# B&R Automation Studio project AS_lab_3
Automation Studio 4.5.2.102

## Configuration Real

CPU 4PP065.0571-P74, AutomationRuntime D4.52, Build 4.1.2, Vc V4.52.0, Safety 1.6

### Task classes (Cpu.sw)
```
Cyclic#1 (cycle 2000 us):
  SDCAxisCtr <- SDCAxisCtrlX.prg
DataObjects: Acp10sys
NcDataObjects: acp10etxen <- acp10etxen.dob, Axis_Xa <- Axis_Xobj.Axis_Xa.dob, Axis_Xi <- Axis_Xobj.Axis_Xi.dob
VcDataObjects: GUI <- GUI.dob
Binaries: TCData, udbdef, ashwd, Role, User, sysconf, ashwac, asfw, arconfig, iomap, Acp10map, acp10cfg
Libraries: Acp10man, Acp10par, NcGlobal, Acp10sdc, AsBrStr, Acp10_MC, brsystem, sys_lib, runtime, Acp10sim, AsIOTime, MotorCtrl, astime, fileio, powerlnk
```

### Hardware
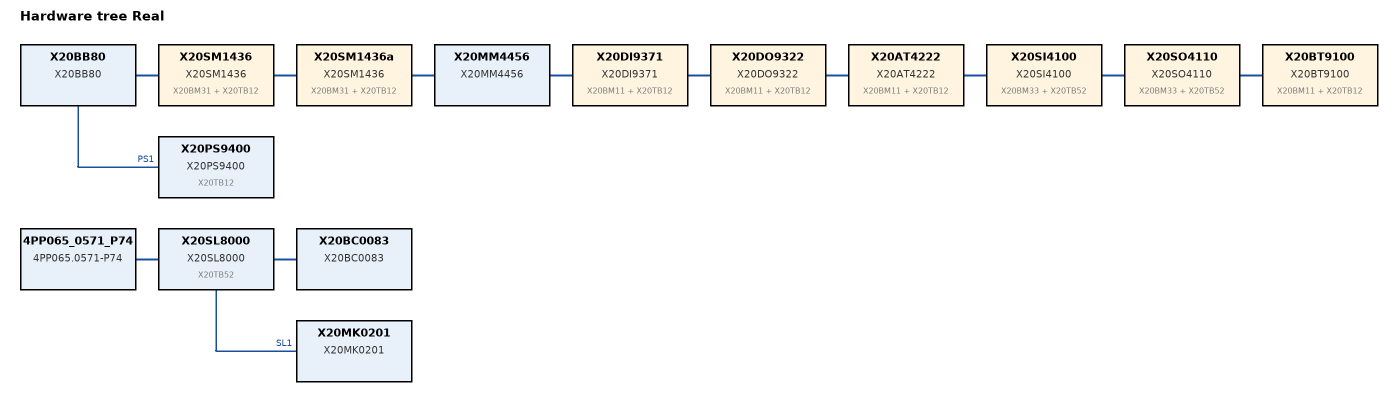
```
4PP065_0571_P74 : 4PP065.0571-P74 v1.1.2.0
  Connector IF5:
    ActivateDevice = 1
    Mode = Manual
    InternetAddress = 10.0.1.10
    SubnetMask = 255.255.255.0
  ConfigurationID = labBR
  TimerDeviceType = EPLX2X
  TimerDevice = 4PP065_0571_P74.IF4
  TaskClassIdleTime = 2000
  Cyclic1Duration = 2000
  Cyclic1Output = 1
  VcObjectName = GUI
X20AT4222 : X20AT4222 v1.2.3.0  [SS1 -> X20TB12e.SS; SL -> X20BM11b.SL1]
X20BB80 : X20BB80 v1.0.2.0
X20BC0083 : X20BC0083 v2.8.0.0  [PLK1 -> X20SL8000.PLK2 [Cable Type=PowerlinkCable, Length=10, Version=1.0.0.2]; SL -> X20BB80.SL1]
X20BM11 : X20BM11 v1.0.0.1  [X2X1 -> X20MM4456.X2X2]
X20BM11a : X20BM11 v1.0.0.1  [X2X1 -> X20BM11.X2X2]
X20BM11b : X20BM11 v1.0.0.1  [X2X1 -> X20BM11a.X2X2]
X20BM11c : X20BM11 v1.0.0.1  [X2X1 -> X20BM33a.X2X2]
X20BM31 : X20BM31 v1.0.0.1  [X2X1 -> X20BB80.IF1]
X20BM31a : X20BM31 v1.0.0.1  [X2X1 -> X20BM31.X2X2]
X20BM33 : X20BM33 v1.0.0.4  [X2X1 -> X20BM11b.X2X2]
X20BM33a : X20BM33 v1.0.0.4  [X2X1 -> X20BM33.X2X2]
X20BT9100 : X20BT9100 v1.0.3.0  [SS1 -> X20TB12f.SS; SL -> X20BM11c.SL1]
X20DI9371 : X20DI9371 v1.0.2.0  [SS1 -> X20TB12c.SS; SL -> X20BM11.SL1]
X20DO9322 : X20DO9322 v1.0.3.0  [SS1 -> X20TB12d.SS; SL -> X20BM11a.SL1]
X20MK0201 : X20MK0201 v1.0.0.0  [SL -> X20SL8000.SL1]
X20MM4456 : X20MM4456 v1.1.5.0  [X2X1 -> X20BM31a.X2X2]
X20PS9400 : X20PS9400 v1.0.2.4  [SS1 -> X20TB12.SS; PS -> X20BB80.PS1]
X20SI4100 : X20SI4100 v1.10.1.1  [SS1 -> X20TB52a.SS; SL -> X20BM33.SL1]
X20SL8000 : X20SL8000 v1.6.5.1  [PLK1 -> 4PP065_0571_P74.IF4 [Cable Type=PowerlinkCable, Length=10, Version=1.0.0.2]; PLK2 -> X20BC0083.PLK1 [Cable Type=PowerlinkCable, Length=10, Version=1.0.0.2]; SS1 -> X20TB52.SS]
  SafeProject = SafeLOGIC-1
X20SM1436 : X20SM1436 v1.4.2.1  [SS1 -> X20TB12a.SS; SL -> X20BM31.SL1]
X20SM1436a : X20SM1436 v1.4.2.1  [SS1 -> X20TB12b.SS; SL -> X20BM31a.SL1]
X20SO4110 : X20SO4110 v1.10.1.1  [SS1 -> X20TB52b.SS; SL -> X20BM33a.SL1]
  SafeModuleID = 3
X20TB12 : X20TB12 v1.0.0.0
X20TB12a : X20TB12 v1.0.0.0
X20TB12b : X20TB12 v1.0.0.0
X20TB12c : X20TB12 v1.0.0.0
X20TB12d : X20TB12 v1.0.0.0
X20TB12e : X20TB12 v1.0.0.0
X20TB12f : X20TB12 v1.0.0.0
X20TB52 : X20TB52 v1.0.0.1
X20TB52a : X20TB52 v1.0.0.1
X20TB52b : X20TB52 v1.0.0.1
```

### IoMap.iom - 4PP065_0571_P74/IoMap.iom
```iecst
VAR_CONFIG
	::SDCAxisCtr:pwm_period AT %QW."X20MM4456".PeriodDurationPWM;
	::SDCAxisCtr:axis_X.pwm_value AT %QW."X20MM4456".PulseWidthCurrentPWM01;
	::SDCAxisCtr:axis_X.reset_error AT %QX."X20MM4456".ClearError01;
	::SDCAxisCtr:axis_X.reset_counter AT %QX."X20MM4456".ResetCounter01;
	::SDCAxisCtr:axis_X.counter AT %IW."X20MM4456".Counter01;
	::SDCAxisCtr:axis_X.endswitch_a_reached AT %IX."X20MM4456".StatusInput03;
	::SDCAxisCtr:axis_X.endswitch_b_reached AT %IX."X20MM4456".StatusInput04;
	::SDCAxisCtr:coil_pwm_value AT %QW."X20MM4456".PulseWidthCurrentPWM04;
END_VAR
```

### Acp10map1.ncm - 4PP065_0571_P74/Motion/Acp10map1.ncm
```
NcMapping (NcSwId=ACP10, DisabledNodesAreHidden=False)
  NcObject Axis_X (ModuleAddress=SDC_IF1.ST2, InterfaceType=SDC, Type=ncAXIS, Channel=1, InitParameter=Axis_Xi, AcoposParameter=Axis_Xa, Disabled=FALSE, ModuleDisabled=FALSE)
```

### Acp10map.ncm - 4PP065_0571_P74/Package/Acp10map.ncm
```
NcMapping (NcSwId=Acp10)
  NcObject X20SM1436_ncAXIS1 (ModuleId=X20SM1436, ModuleAddress=SDC_IF1.ST1, Type=ncAXIS, Channel=1, AcoposSimulation=Off, Disabled=TRUE, ModuleDisabled=FALSE)
  NcObject X20SM1436a_ncAXIS1 (ModuleId=X20SM1436a, ModuleAddress=SDC_IF1.ST2, Type=ncAXIS, Channel=1, AcoposSimulation=Off, Disabled=TRUE, ModuleDisabled=FALSE)
  NcObject 8I64xxxxxxx.00x-1_ncAXIS1 (ModuleId=8I64xxxxxxx.00x-1, ModuleAddress=SDC_IF1.ST3, Type=ncAXIS, Channel=1, AcoposSimulation=Off, Disabled=TRUE, ModuleDisabled=FALSE)
```

## Logical view

Binary libraries used (declarations not repeated): operator, runtime, astime, AsIecCon, Acp10man, Acp10par, NcGlobal, Acp10sdc, AsBrStr, Acp10_MC, brsystem, sys_lib, Acp10sim, AsIOTime

### Global.var - Global variables
```iecst
VAR
	Axis_X : ACP10AXIS_typ;
	Axis_X_HW : SdcHwCfg_typ;
	Axis_X_EncIf : SdcEncIf16_typ;
	Axis_X_DrvIf : SdcDrvIf16_typ;
	Axis_X_DiDoIf : SdcDiDoIf_typ;
END_VAR
```

### Package Logical/Libraries - Global libraries

### Library Logical/Libraries/MotorCtrl (ANSIC)

#### MotorCtrl.fun
```iecst
FUNCTION_BLOCK FB_Regulator
	VAR_INPUT
		e : REAL;
		e_prev : REAL;
	END_VAR
	VAR_OUTPUT
		u : REAL;
	END_VAR
	VAR
		u_raw : REAL;
		k_p : REAL;
		k_i : REAL;
		integrator : FB_Integrator;
		iyOld : REAL;
		max_abs_value : REAL;
	END_VAR
END_FUNCTION_BLOCK

FUNCTION_BLOCK FB_Motor
	VAR_INPUT
		u : REAL;
	END_VAR
	VAR_OUTPUT
		w : REAL;
		phi : REAL;
	END_VAR
	VAR
		integrator : FB_Integrator;
		integrator_phi : FB_Integrator;
		Tm : REAL;
		ke : REAL;
		enable_reg : BOOL;
	END_VAR
END_FUNCTION_BLOCK

FUNCTION_BLOCK FB_Integrator
	VAR_INPUT
		in : REAL;
	END_VAR
	VAR_OUTPUT
		out : REAL;
	END_VAR
	VAR
		dt : REAL;
		direct : BOOL;
	END_VAR
END_FUNCTION_BLOCK

FUNCTION_BLOCK FB_Axis
	VAR_INPUT
		u : REAL;
		force_a : BOOL;
		force_b : BOOL;
		endswitch_a_reached : BOOL;
		endswitch_b_reached : BOOL;
	END_VAR
	VAR_OUTPUT
		reset_error : BOOL;
		reset_counter : BOOL;
		pwm_value : INT;
		counter : INT;
		speed : INT;
	END_VAR
	VAR
		last_counter : INT;
		ForceStop : BOOL;
		Home : BOOL;
	END_VAR
END_FUNCTION_BLOCK
```

#### FB_Axis.c
```c
#include <bur/plctypes.h>
#ifdef __cplusplus
	extern "C"
	{
#endif
#include "MotorCtrl.h"
#ifdef __cplusplus
	};
#endif
/* TODO: Add your comment here */
void FB_Axis(struct FB_Axis* inst)
{
	if (inst->Home)
	{
		inst->pwm_value = 0;
		inst->reset_counter = 1;
		inst->Home = 0;
	}

	if (!inst->ForceStop)
	{
		if (inst->endswitch_a_reached && inst->u < 0)
		{
			inst->pwm_value = 0;
			inst->reset_error = 1;
		}
		else if (inst->endswitch_b_reached && inst->u > 0)
		{
			inst->pwm_value = 0;
			inst->reset_error = 1;
		}
		else if (inst->force_a)
		{
			inst->pwm_value = 0;
			inst->endswitch_a_reached = inst->force_a;
		}
		else if (inst->force_b)
		{
			inst->pwm_value = 0;
			inst->endswitch_b_reached = inst->force_b;
		}
		else
		{
			inst->pwm_value = inst->u / 24.0 * 32767;
			inst->reset_error = 0;
		}
	}
	else
	{
		inst->pwm_value = 0;
	}

	inst->speed = inst->u / 24.0 * 6500;
}
```

#### FB_Regulator.c
```c
#include <bur/plctypes.h>
#ifdef __cplusplus
	extern "C"
	{
#endif
#include "MotorCtrl.h"
#ifdef __cplusplus
	};
#endif

#include "Math.h"
/* TODO: Add your comment here */
void FB_Regulator(struct FB_Regulator* inst)
{
	if (inst->integrator.direct)
		inst->integrator.in = inst->k_i * inst->e_prev + inst->iyOld / inst->integrator.dt;
	else
		inst->integrator.in = inst->k_i * inst->e + inst->iyOld / inst->integrator.dt;
	FB_Integrator(&inst->integrator);
	inst->u_raw = (fabs(inst->k_p * inst->e) < inst->max_abs_value ? inst->k_p * inst->e : inst->max_abs_value * copysign(1.0, inst->k_p * inst->e)) +
		inst->integrator.out;
	inst->u = fabs(inst->u_raw) < inst->max_abs_value ? inst->u_raw : inst->max_abs_value * copysign(1.0, inst->u_raw);
	inst->iyOld = inst->u - inst->u_raw;
}
```

### Package Logical/Axis_Xobj - Axis_Xobj

### Axis_Xi.ax
```
InitParameter (Version=5.02.1, NcSwId=Acp10)
  ACP10AXIS_typ:
    dig_in:
      level:
        reference = ncACTIV_HI
        pos_hw_end = ncACTIV_HI
        neg_hw_end = ncACTIV_HI
        trigger1 = ncACTIV_HI
        trigger2 = ncACTIV_LO + ncQUICKSTOP
    encoder_if:
      parameter:
        count_dir = ncSTANDARD
        scaling:
          load:
            units = 3000
            rev_motor = 1
    limit:
      parameter:
        v_pos = 10000
        v_neg = 10000
        a1_pos = 10000.0
        a2_pos = 10000.0
        a1_neg = 10000.0
        a2_neg = 10000.0
        t_jolt = 0
        t_in_pos = 0
        pos_sw_end = 2000000000
        neg_sw_end = -2000000000
        ds_warning = 500
        ds_stop = 50000.0
        a_stop = 1.0e30
        dv_stop = 0
        dv_stop_mode = ncOFF
    controller:
      mode = ncPOSITION
      position:
        kv = 10.0
        tn = 0
        t_predict = 0.0004
        t_total = 0.0004
        p_max = 1.0e30
        i_max = 0
      speed:
        kv = 2.0
        tn = 0
        t_filter = 0.0
        isq_filter1:
          type = ncOFF
          a0 = 0.0
          a1 = 0.0
          b0 = 0.0
          b1 = 0.0
          b2 = 0.0
          c0_par_id = 0
          c1_par_id = 0
        isq_filter2:
          type = ncOFF
          a0 = 0.0
          a1 = 0.0
          b0 = 0.0
          b1 = 0.0
          b2 = 0.0
          c0_par_id = 0
          c1_par_id = 0
        isq_filter3:
          type = ncOFF
          a0 = 0.0
          a1 = 0.0
          b0 = 0.0
          b1 = 0.0
          b2 = 0.0
          c0_par_id = 0
          c1_par_id = 0
      uf:
        type = ncLINEAR + ncCORRECTION
        auto_config = ncMOTOR_PAR
        u0 = 0
        un = 0
        fn = 50.0
        k_f_slip = 0
      ff:
        torque_load = 0.0
        torque_pos = 0.0
        torque_neg = 0.0
        kv_torque = 0.0
        inertia = 0.0
        t_filter_a = 0.0
    move:
      stop:
        parameter[0]:
          decel_ramp = ncA_LIMIT
          controller = ncON
        parameter[1]:
          decel_ramp = ncA_LIMIT
          controller = ncON
        parameter[2]:
          decel_ramp = ncA_LIMIT
          controller = ncON
        parameter[3]:
          decel_ramp = ncA_LIMIT
          controller = ncON
        quickstop:
          decel_ramp = ncA_LIMIT
          t_jolt = 0
        drive_error:
          decel_ramp = ncA_LIMIT
      homing:
        parameter:
          s = 0
          v_switch = 6000.0
          v_trigger = 2000.0
          a = 10000.0
          mode = ncEND_SWITCH
          edge_sw = ncNEGATIVE
          start_dir = ncPOSITIVE
          trigg_dir = ncNEGATIVE
          ref_pulse = ncOFF
          fix_dir = ncOFF
          tr_s_block = 0
          torque_lim = 0
          ds_block = 0
          ds_stop = 0
      basis:
        parameter:
          v_pos = 5000
          v_neg = 5000
          a1_pos = 50000
          a2_pos = 50000
          a1_neg = 50000
          a2_neg = 50000
    message:
      text:
        parameter:
          format = ncBREAK
          columns = 80
          data_modul = acp10etxen
```

### Program Logical/SDCAxisCtrlX (ANSIC)

#### Variables.var
```iecst
VAR
	axis_X : FB_Axis;
	CoilPowered : BOOL;
	CoilPWM : INT;
	fb_regulator : FB_Regulator;
	PWM_Period : UINT;
END_VAR
```

#### Main.c
```c
/*#include <bur/plctypes.h>
#include <math.h>

#ifdef _DEFAULT_INCLUDES
	#include <AsDefault.h>
#endif

#define MOTORS_COUNT 3

void _INIT MainINIT(void)
{
	//Устанавливаем типы SDC модулей
	Axis_X_HW.EncIf1_Typ = ncSDC_ENC16;
	Axis_X_HW.DiDoIf_Typ = ncSDC_DIDO;
	Axis_X_HW.DrvIf_Typ = ncSDC_DRVSERVO16;
	//Устанавливаем имена переменных
	strcpy(Axis_X_HW.EncIf1_Name, "Axis_X_EncIf");
	strcpy(Axis_X_HW.DrvIf_Name, "Axis_X_DrvIf");
	strcpy(Axis_X_HW.DiDoIf_Name, "Axis_X_DiDoIf");
	//Устанавливаем входы готовности и нормальной
	работы
	Axis_X_EncIf.iEncOK = 1;
	Axis_X_DrvIf.iDrvOK = 1;
	Axis_X_DrvIf.iStatusEnable = 1;
	Axis_X_DiDoIf.iDriveReady = 1;

	Axis_X_EncIf.iLifeCnt++;
	Axis_X_DiDoIf.iLifeCntDriveEnable++;
	Axis_X_DiDoIf.iLifeCntDriveReady++;
	Axis_X_DiDoIf.iLifeCntNegHwEnd++;
	Axis_X_DiDoIf.iLifeCntPosHwEnd++;
	Axis_X_DiDoIf.iLifeCntReference++;
	Axis_X_DrvIf.iLifeCnt++;
	Axis_X_EncIf.iActTime = (INT)AsIOTimeCyclicStart();

	int i = 0;
	for (; i < MOTORS_COUNT; i++)
	{
		motors[i].pwm_value = 0;
		motors[i].pwm_percentage = 0;
		motors[i].counter = 0;
		motors[i].coordinate = 0;
		motors[i].button_status = 0;
		motors[i].reset_error = 0;
		motors[i].endswitch_a_reached = 0;
		motors[i].endswitch_b_reached = 0;
	}
	pwm_period = 200;
	coil_powered = 0;
	coil_pwm_value = 0;
	emergency_stop = 0;
	current_motor_index = 0;

	check = 0;
	a = 0;
	n = 0;
}

void _CYCLIC MainCYCLIC(void)
{
	int i = 0, j = 0;
	if (emergency_stop)  //аварийная остановка
	{
		for (i = 0; i < MOTORS_COUNT; i++)
		{
			motors[i].pwm_value = 0;
			motors[i].pwm_percentage = 0;
		}
		coil_powered = 0;
		check = 0;
		emergency_stop = 0;
	}
	current_motor = &motors[current_motor_index];
	for (i = 0; i < MOTORS_COUNT; i++)  //цикл для обозначения на экране текущей степени (кнопка подсвечивается белым цветом)
	{
		MotorFunctionBlock(&motors[i]);
		if (current_motor == &motors[i])
		{
			motors[i].button_status = 1 << 1;
		}
		else
		{
			motors[i].button_status = 0;
		}
	}
	if (coil_powered)  //проверяем напряжение на катушке
	{
		coil_pwm_value = 32767;
		if (check)
		{
			switch (mode)  //проверяем выбранный режим
			{
				case 1:
					switch (path)  //проверяем выбранный контур, разбиваем его и заполняем массив координат соответствующими значениями
					{
						case 1:
							for (i = 0; i < 20; i++)
							{
								coordX[i] = 150 * pi * i / (10*sqrt(2));
								coordY[i] = 150 * pi * i / (10*sqrt(2));
								coordZ[i] = 250 * sin(sqrt(coordX[i] * coordX[i] + coordY[i] * coordY[i]) / 150);
							}
							break;
						case 2:
							for (i = 0; i < 20; i++)
							{
								coordX[i] = 30 * i;
								coordY[i] = 30 * i;
								coordZ[i] = (coordX[i] * coordX[i] + coordY[i] * coordY[i]) / 180;
							}
							break;
						case 0:
							break;
					}
					distX = coordX[a+1] - coordX[a];  //длина полученных отрезков
					distY = coordY[a+1] - coordY[a];
					distZ = coordZ[a+1] - coordZ[a];
					if ((fabs(distX) >= fabs(distY)) && (fabs(distX) >= fabs(distZ)))  //поиск наибольшей проекции каждого отрезка
					{
						index[a] = 2;
					}
					if ((fabs(distY) >= fabs(distX)) && (fabs(distY) >= fabs(distZ)))
					{
						index[a] = 0;
					}
					if ((fabs(distZ) >= fabs(distX)) && (fabs(distZ) >= fabs(distY)))
					{
						index[a] = 1;
					}
					if (index[a] == 2)  //проекция на ось X наибольшая
					{
						if (motors[2].counter > coordX[a+1])  //если степень находится за следующей точкой, то двигаем её в обратном направлении
						{
							motors[2].pwm_percentage_float = -50.0;
						}
						if (motors[2].counter < coordX[a+1])  //если перед точкой, то в прямом направлении
						{
							motors[2].pwm_percentage_float = 50.0;
						}
						motors[0].pwm_percentage_float = (distY * motors[2].pwm_percentage_float) / distX;  //вычисляем реальное значение ШИМ (в процентах)
						motors[1].pwm_percentage_float = (distZ * motors[2].pwm_percentage_float) / distX;
						if ((motors[2].counter >= (coordX[a+1] - 2)) && (motors[2].counter <= (coordX[a+1] + 2)))
						{
							if (a < 18)  //проверка пройденных точек
							{
								a++;
							}
							else  //если все точки пройдены, то отключаем степени и сбрасываем выбранные режим и контур
							{
								for (i = 0; i < MOTORS_COUNT; i++)
								{
									motors[i].pwm_percentage_float = 0.0;
									motors[i].pwm_value_float = 0.0;
									motors[i].pwm_percentage = 0;
									motors[i].pwm_value = 0;
								}
								check = 0;
								mode = 0;
								path = 0;
								a = 0;
							}
						}
					}
					if (index[a] == 0)  //проекция на ось Y максимальная
					{
						if (motors[0].counter > coordY[a+1])  //если степень находится за следующей точкой, то двигаем её в обратном направлении
						{
							motors[0].pwm_percentage_float = -50.0;
						}
						if (motors[0].counter < coordY[a+1])  //если перед точкой, то в прямом направлении
						{
							motors[0].pwm_percentage_float = 50.0;
						}
						motors[2].pwm_percentage_float = (distX * motors[0].pwm_percentage_float) / distY;  //вычисляем реальное значение ШИМ (в процентах)
						motors[1].pwm_percentage_float = (distZ * motors[0].pwm_percentage_float) / distY;
						if ((motors[0].counter >= (coordY[a+1] - 2)) && (motors[0].counter <= (coordY[a+1] + 2)))
						{
							if (a < 18)  //проверка пройденных точек
							{
								a++;
							}
							else  //если все точки пройдены, то отключаем степени и сбрасываем выбранные режим и контур
							{
								for (i = 0; i < MOTORS_COUNT; i++)
								{
									motors[i].pwm_percentage_float = 0.0;
									motors[i].pwm_value_float = 0.0;
									motors[i].pwm_percentage = 0;
									motors[i].pwm_value = 0;
								}
								check = 0;
								mode = 0;
								path = 0;
								a = 0;
							}
						}
					}
					if (index[a] == 1)  //проекция на ось Z максимальная
					{
						if (motors[1].counter > coordZ[a+1])  //если степень находится за следующей точкой, то двигаем её в обратном направлении
						{
							motors[1].pwm_percentage_float = -50.0;
						}
						if (motors[1].counter < coordZ[a+1])  //если перед точкой, то в прямом направлении
						{
							motors[1].pwm_percentage_float = 50.0;
						}
						motors[2].pwm_percentage_float = (distX * motors[1].pwm_percentage_float) / distZ;  //вычисляем реальное значение ШИМ (в процентах)
						motors[0].pwm_percentage_float = (distY * motors[1].pwm_percentage_float) / distZ;
						if ((motors[1].counter >= (coordZ[a+1] - 2)) && (motors[1].counter <= (coordZ[a+1] + 2)))
						{
							if (a < 18)  //проверка пройденных точек
							{
								a++;
							}
							else  //если все точки пройдены, то отключаем степени и сбрасываем выбранные режим и контур
							{
								for (i = 0; i < MOTORS_COUNT; i++)
								{
									motors[i].pwm_percentage_float = 0.0;
									motors[i].pwm_value_float = 0.0;
									motors[i].pwm_percentage = 0;
									motors[i].pwm_value = 0;
								}
								check = 0;
								mode = 0;
								path = 0;
								a = 0;
							}
						}
					}
					for (i = 0; i < MOTORS_COUNT; i++)
					{
						motors[i].pwm_percentage = motors[i].pwm_percentage_float;  //присваиваем значению ШИМ на слайдере на экране к реальному значению ШИМ (для наглядности)
					}
					for (i = 0; i < MOTORS_COUNT; i++)
					{
						motors[i].pwm_value_float = 32767 * motors[i].pwm_percentage_float / 100;  //вычисляем ШИМ для каждой степени
						motors[i].pwm_value = motors[i].pwm_value_float;  //приводим значение типа REAL к значению типа INT и пересылаем на двигатель
						if ((!motors[i].endswitch_a_reached) && (!motors[i].endswitch_b_reached))
						{
							motors[i].reset_error = 0;
						}
						if ((motors[i].endswitch_a_reached) && (motors[i].pwm_percentage > 0))  //если достигнут концевой датчик, то останавливаем все степени и сбрасываем ошибку
						{
							motors[i].reset_error = 1;
							for (j = 0; j < MOTORS_COUNT; j++)
							{
								motors[j].pwm_percentage_float = 0.0;
								motors[j].pwm_value_float = 0.0;
								motors[j].pwm_percentage = 0;
								motors[j].pwm_value = 0;
							}
						}
						if ((motors[i].endswitch_b_reached) && (motors[i].pwm_percentage < 0))
						{
							motors[i].reset_error = 1;
							for (j = 0; j < MOTORS_COUNT; j++)
							{
								motors[j].pwm_percentage_float = 0.0;
								motors[j].pwm_value_float = 0.0;
								motors[j].pwm_percentage = 0;
								motors[j].pwm_value = 0;
							}
						}
					}
					break;  //закрытие 1-го режима
				case 2:
					switch (path)  //проверяем выбранный контур и задаем соответствующие функции изменения скоростей движения степеней
					{
						case 1:
							motors[0].pwm_percentage_float = 50.0;
							motors[2].pwm_percentage_float = 50.0;
							motors[1].pwm_percentage_float = 90 * cos(pi * n / 40);
							break;
						case 2:
							motors[0].pwm_percentage_float = 50.0;
							motors[2].pwm_percentage_float = 50.0;
							if ((n * n / 60) <= 100)  //ШИМ не может быть больше 100%
							{
								motors[1].pwm_percentage_float = n * n / 60;
							}
							else  //если больше 100%, то отключаем степени и сбрасываем выбранные режим и контур
							{
								for (i = 0; i < MOTORS_COUNT; i++)
								{
									motors[i].pwm_percentage_float = 0.0;
									motors[i].pwm_value_float = 0.0;
									motors[i].pwm_percentage = 0;
									motors[i].pwm_value = 0;
								}
								check = 0;
								mode = 0;
								path = 0;
								n = 0;
							}
						case 0:
							break;
					}
					if (n < 80)  //за 1 секунду проходит 10 итераций основного цикла; если движение происходит 8 секунд, то к концу 8-ой секунды пройдет 80 итераций
					{
					n++;
					}
					else  //если все итерации пройдены, то отключаем степени и сбрасываем выбранные режим и контур
					{
					for (i = 0; i < MOTORS_COUNT; i++)
					{
					motors[i].pwm_percentage_float = 0.0;
					motors[i].pwm_value_float = 0.0;
					motors[i].pwm_percentage = 0;
					motors[i].pwm_value = 0;
					}
					check = 0;
					mode = 0;
					path = 0;
					n = 0;
					}
					for (i = 0; i < MOTORS_COUNT; i++)
					{
						motors[i].pwm_percentage = motors[i].pwm_percentage_float;  //присваиваем значению ШИМ на слайдере на экране к реальному значению ШИМ (для наглядности)
					}
					for (i = 0; i < MOTORS_COUNT; i++)
					{
						motors[i].pwm_value_float = 32767 * motors[i].pwm_percentage_float / 100;  //вычисляем ШИМ для каждой степени
						motors[i].pwm_value = motors[i].pwm_value_float;  //приводим значение типа REAL к значению типа INT и пересылаем на двигатель
						if ((!motors[i].endswitch_a_reached) && (!motors[i].endswitch_b_reached))
						{
							motors[i].reset_error = 0;
						}
						if ((motors[i].endswitch_a_reached) && (motors[i].pwm_percentage > 0))  //если достигнут концевой датчик, то останавливаем все степени и сбрасываем ошибку
						{
							motors[i].reset_error = 1;
							for (j = 0; j < MOTORS_COUNT; j++)
							{
								motors[j].pwm_percentage_float = 0.0;
								motors[j].pwm_value_float = 0.0;
								motors[j].pwm_percentage = 0;
								motors[j].pwm_value = 0;
							}
						}
						if ((motors[i].endswitch_b_reached) && (motors[i].pwm_percentage < 0))
						{
							motors[i].reset_error = 1;
							for (j = 0; j < MOTORS_COUNT; j++)
							{
								motors[j].pwm_percentage_float = 0.0;
								motors[j].pwm_value_float = 0.0;
								motors[j].pwm_percentage = 0;
								motors[j].pwm_value = 0;
							}
						}
					}
					break;  //закрытие 2-го режима
				case 0:
					break;
			}
		}
		else  //если движение не начато, то переходим в режим ручного управления через сенсорный экран (для отладки, приведения в начало координат и т.д.)
		{
			for (i = 0; i < MOTORS_COUNT; i++)
			{
				motors[i].pwm_value = 32767 * motors[i].pwm_percentage / 100;
				if ((!motors[i].endswitch_a_reached) && (!motors[i].endswitch_b_reached))
				{
					motors[i].reset_error = 0;
				}
				if ((motors[i].endswitch_a_reached) && (motors[i].pwm_percentage > 0))
				{
					motors[i].reset_error = 1;
					motors[i].pwm_percentage = 0;
					motors[i].pwm_value = 0;
				}
				if ((motors[i].endswitch_b_reached) && (motors[i].pwm_percentage < 0))
				{
					motors[i].reset_error = 1;
					motors[i].pwm_percentage = 0;
					motors[i].pwm_value = 0;
				}
			}
		}
	}
	else  //если нет напряжения на катушке, то отключаем все степени
	{
		coil_pwm_value = 0;
		for (i = 0; i < MOTORS_COUNT; i++)
		{
			motors[i].pwm_value = 0;
		}
	}
}

void _EXIT ProgramExit(void)
{

}*/

#include <bur/plctypes.h>

#ifdef _DEFAULT_INCLUDES
#include <AsDefault.h>
#endif

void increase_counters(void);

void _INIT ProgramInit(void)
{
	//Устанваливаем типы SDC модулей
	Axis_X_HW.EncIf1_Typ = ncSDC_ENC16;
	Axis_X_HW.DiDoIf_Typ = ncSDC_DIDO;
	Axis_X_HW.DrvIf_Typ = ncSDC_DRVSERVO16;

	//Устанавливаем имена переменных
	strcpy(Axis_X_HW.EncIf1_Name, "Axis_X_EncIf");
	strcpy(Axis_X_HW.DrvIf_Name, "Axis_X_DrvIf");
	strcpy(Axis_X_HW.DiDoIf_Name, "Axis_X_DiDoIf");

	//Устанавливаем входы готовности и нормальной работы
	Axis_X_EncIf.iEncOK = 1;
	Axis_X_DrvIf.iDrvOK = 1;
	Axis_X_DrvIf.iStatusEnable = 1;
	Axis_X_DiDoIf.iDriveReady = 1;

	fb_regulator.integrator.dt = 0.002;
	fb_regulator.integrator.direct = 0;
	fb_regulator.k_i = 0.16;
	fb_regulator.k_p = 0.0064;
	fb_regulator.max_abs_value = 12.0;

	pwm_period = 200;
}

void _CYCLIC ProgramCyclic(void)
{
	increase_counters();
	Axis_X_EncIf.iActTime = (INT)	AsIOTimeCyclicStart();

	Axis_X_EncIf.iActPos = axis_X.counter;
	Axis_X_DiDoIf.iPosHwEnd = axis_X.endswitch_b_reached;
	Axis_X_DiDoIf.iNegHwEnd = axis_X.endswitch_a_reached;

	if (coil_powered)
	{
		coil_pwm_value = 32767;

		fb_regulator.e = Axis_X_DrvIf.oSetPos - axis_X.speed;
		FB_Regulator(&fb_regulator);

		axis_X.u = fb_regulator.u;
		FB_Axis(&axis_X);
	}
	else
	{
		coil_pwm_value = 0;

		fb_regulator.e = -axis_X.speed;
		FB_Regulator(&fb_regulator);

		axis_X.u = fb_regulator.u;
		FB_Axis(&axis_X);
	}
}

void increase_counters(void)
{
	Axis_X_EncIf.iLifeCnt++;
	Axis_X_DiDoIf.iLifeCntDriveEnable++;
	Axis_X_DiDoIf.iLifeCntDriveReady++;
	Axis_X_DiDoIf.iLifeCntNegHwEnd++;
	Axis_X_DiDoIf.iLifeCntPosHwEnd++;
	Axis_X_DiDoIf.iLifeCntReference++;
	Axis_X_DrvIf.iLifeCnt++;
}

void _EXIT ProgramExit(void)
{
	// Insert code here

}
```

- Visualisation Logical/GUI (not shown)

### Program Logical/SDCCTRL

#### Main.c
```c
#include <bur/plctypes.h>

#ifdef _DEFAULT_INCLUDES
	#include <AsDefault.h>
#endif

void _INIT ProgramInit(void)
{
	//Устанваливаем типы SDC модулей
	Axis_X_HW.EncIf1_Typ = ncSDC_ENC16;
	Axis_X_HW.DiDoIf_Typ = ncSDC_DIDO;
	Axis_X_HW.DrvIf_Typ = ncSDC_DRVSERVO16;

	//Устанавливаем имена переменных
	strcpy(Axis_X_HW.EncIf1_Name, "Axis_X_EncIf");
	strcpy(Axis_X_HW.DrvIf_Name, "Axis_X_DrvIf");
	strcpy(Axis_X_HW.DiDoIf_Name, "Axis_X_DiDoIf");

	//Устанавливаем входы готовности и нормальной работы
	Axis_X_EncIf.iEncOK = 1;
	Axis_X_DrvIf.iDrvOK = 1;
	Axis_X_DrvIf.iStatusEnable = 1;
	Axis_X_DiDoIf.iDriveReady = 1;
}

void _CYCLIC ProgramCyclic(void)
{
	Axis_X_EncIf.iLifeCnt++;
	Axis_X_DiDoIf.iLifeCntDriveEnable++;
	Axis_X_DiDoIf.iLifeCntDriveReady++;
	Axis_X_DiDoIf.iLifeCntNegHwEnd++;
	Axis_X_DiDoIf.iLifeCntPosHwEnd++;
	Axis_X_DiDoIf.iLifeCntReference++;
	Axis_X_DrvIf.iLifeCnt++;

	Axis_X_EncIf.iActTime = (INT)	AsIOTimeCyclicStart();
}

void _EXIT ProgramExit(void)
{

}
```

Listed in the project but not available here: Logical/Global.typ, Logical/acp10etxen
